// TIA Portal V18 export
DATA_BLOCK "MachineDB"   // DB22
{ S7_Optimized_Access := 'FALSE' }
VERSION : 0.1
// stored: AutoNumber true, DBAccessibleFromOPCUA true, IsOnlyStoredInLoadMemory false, IsWriteProtectedInAS false
   VAR RETAIN
      SerialNumber : Int := 2011;
      AutomateVersion : Int := 6;
      MachineType { ExternalWritable := 'False'} : String := 'ArmadilloV7BR';   // Not writable from HMI
      MachineLimit : Struct
         XSafety : Struct
            PosMax : DInt := 0;
            PosMin : DInt := 0;
            SafetyMargin : DInt;
            VelocityMax : DInt;
            VelocityMin : DInt;
         END_STRUCT;
         YSafety : Struct
            PosMax : DInt := 0;
            PosMin : DInt := 0;
            SafetyMargin : DInt;
            VelocityMax : DInt;
            VelocityMin : DInt;
         END_STRUCT;
         Z1Safety : Struct
            PosMax : DInt := 0;
            PosMin : DInt := 0;
            SafetyMargin : DInt;
            VelocityMax : DInt;
            VelocityMin : DInt;
         END_STRUCT;
         Z2Safety : Struct
            PosMax : DInt := 0;
            PosMin : DInt := 0;
            SafetyMargin : DInt;
            VelocityMax : DInt;
            VelocityMin : DInt;
         END_STRUCT;
         Heater : Struct
            FeedboxStart : DInt;
            FeedboxEnd : DInt;
            PrintboxStart : DInt;
            PrintboxEnd : DInt;
         END_STRUCT;
      END_STRUCT;
      ArmadilloOption : Struct
         MachineTypeNext : String := 'ArmadilloV7BR';
         DoorOption { ExternalWritable := 'False'} : Int := 3;   // SAFETY OPTION, ASK BEFORE CHANGING
         DoorOptionNext : Int := 3;
         DepowderingBox : Int;   // 0 if no box; 1 is we use V1 of the box;
         DepowderingBoxNext : Int;   // 0 if no box; 1 is we use V1 of the box;
         ZAxisDriveOption : String := 'CMMT';   // CMMT;CMMS;
         ZAxisDriveOptionNext : String := 'CMMT';   // CMMT;CMMS;
         UVOption : Int := 1;   // 0 means no UV lamp; 1 version of the UV lamp;
         UVOptionNext : Int := 1;   // 0 means no UV lamp; 1 version of the UV lamp;
         StacklightOption : Int := 1;   // 0 means no Stacklight; 1 version of the Stacklight;
         StacklightOptionNext : Int := 1;   // 0 means no Stacklight; 1 version of the Stacklight;
         CappingStationOption : Int := 1;   // 0 means no Capping Station; 1 version of the Capping Station;
         CappingStationOptionNext : Int := 1;   // 0 means no Capping Station; 1 version of the Capping Station;
      END_STRUCT;
      MachineLimitSecondary : Struct
         NoGoZone01 : Struct   // Temporary not used -> go to DepowderingBoxDimensions
            NoGoZone01_Xstart : DInt;   // Start of the No Go Zone for Depowdering Box
            NoGoZone01_Xend : DInt;   // Start of the No Go Zone for Depowdering Box
            NoGoZone01_Ystart : DInt;   // Start of the No Go Zone for Depowdering Box
            NoGoZone01_Yend : DInt;   // End of the No Go Zone for Depowdering Box
            NoGoZone01_Z1start : DInt;   // Start of the No Go Zone for Depowdering Box
            NoGoZone01_Z1end : DInt;   // End of the No Go Zone for Depowdering Box
            NoGoZone01_Z2start : DInt;   // Start of the No Go Zone for Depowdering Box
            NoGoZone01_Z2end : DInt;   // End of the No Go Zone for Depowdering Box
         END_STRUCT;
      END_STRUCT;
      MachineTypeString : Struct
         _sArmadilloDev { ExternalWritable := 'False'} : String := 'ArmadilloDev';   // Not writable from HMI
         _sArmadilloV2 { ExternalWritable := 'False'} : String := 'ArmadilloV2';   // Not writable from HMI
         _sArmadilloBRV2 { ExternalWritable := 'False'} : String := 'ArmadilloBRV2';   // Not writable from HMI
         _sArmadilloXLV2 { ExternalWritable := 'False'} : String := 'ArmadilloXLV2';   // Not writable from HMI
         _sArmadilloXLBRV2 { ExternalWritable := 'False'} : String := 'ArmadilloXLBRV2';   // Not writable from HMI
         _sArmadilloV6 { ExternalWritable := 'False'} : String := 'ArmadilloV6';   // Machine 2007;
         _sArmadilloV6BR { ExternalWritable := 'False'} : String := 'ArmadilloV6BR';   // Machine 2007;
         _sArmadilloV7 : String := 'ArmadilloV7';   // Machine 2009; 2011;
         _sArmadilloV7BR : String := 'ArmadilloV7BR';   // Machine 2009; 2011;
         _sArmadilloXLV7 : String := 'ArmadilloXLV7';   // Machine 2010;
         _sArmadilloXLV7BR : String := 'ArmadilloXLV7BR';   // Machine 2010;
      END_STRUCT;
      ArmadilloDevMachine : Struct   // Software limit for the Armadillo Dev machine
         XSafety : Struct
            PosMax : DInt := 454000;
            PosMin : DInt := -3000;
            SafetyMargin : DInt := 0;
            VelocityMax : DInt := 500;
            VelocityMin : DInt := 0;
         END_STRUCT;
         YSafety : Struct
            PosMax : DInt := 1100000;
            PosMin : DInt := -3000;
            SafetyMargin : DInt := 0;
            VelocityMax : DInt := 500;
            VelocityMin : DInt;
         END_STRUCT;
         Z1Safety : Struct
            PosMax : DInt := 297850;
            PosMin : DInt := -3000;
            SafetyMargin : DInt := 0;
            VelocityMax : DInt := 20;
            VelocityMin : DInt;
         END_STRUCT;
         Z2Safety : Struct
            PosMax : DInt := 297850;
            PosMin : DInt := -3000;
            SafetyMargin : DInt := 0;
            VelocityMax : DInt := 20;
            VelocityMin : DInt;
         END_STRUCT;
         Heater : Struct
            FeedboxStart : DInt := 100000;
            FeedboxEnd : DInt := 400000;
            PrintboxStart : DInt := 300000;
            PrintboxEnd : DInt := 765000;
         END_STRUCT;
      END_STRUCT;
      ArmadilloBRMachine : Struct   // Software limit for the Armadillo Dev machine
         XSafety : Struct
            PosMax : DInt := 454000;
            PosMin : DInt := -3000;
            SafetyMargin : DInt;
            VelocityMax : DInt;
            VelocityMin : DInt;
         END_STRUCT;
         YSafety : Struct
            PosMax : DInt := 1100000;
            PosMin : DInt := -3000;
            SafetyMargin : DInt;
            VelocityMax : DInt;
            VelocityMin : DInt;
         END_STRUCT;
         Z1Safety : Struct
            PosMax : DInt := 94000;   // v1 = 210500
            PosMin : DInt := -3000;
            SafetyMargin : DInt;
            VelocityMax : DInt;
            VelocityMin : DInt;
         END_STRUCT;
         Z2Safety : Struct
            PosMax : DInt := 94000;   // v1 = 210500
            PosMin : DInt := -3000;
            SafetyMargin : DInt;
            VelocityMax : DInt;
            VelocityMin : DInt;
         END_STRUCT;
         Heater : Struct
            FeedboxStart : DInt;
            FeedboxEnd : DInt;
            PrintboxStart : DInt;
            PrintboxEnd : DInt;
         END_STRUCT;
      END_STRUCT;
      ArmadilloXLMachine : Struct   // Software limit for the Armadillo Production machine
         XSafety : Struct
            PosMax : DInt := 516000;
            PosMin : DInt := -3000;
            SafetyMargin : DInt;
            VelocityMax : DInt;
            VelocityMin : DInt;
         END_STRUCT;
         YSafety : Struct
            PosMax : DInt := 1380000;
            PosMin : DInt := -3000;
            SafetyMargin : DInt;
            VelocityMax : DInt;
            VelocityMin : DInt;
         END_STRUCT;
         Z1Safety : Struct
            PosMax : DInt := 302000;
            PosMin : DInt := -500;
            SafetyMargin : DInt;
            VelocityMax : DInt;
            VelocityMin : DInt;
         END_STRUCT;
         Z2Safety : Struct
            PosMax : DInt := 302000;
            PosMin : DInt := -500;
            SafetyMargin : DInt;
            VelocityMax : DInt;
            VelocityMin : DInt;
         END_STRUCT;
         Heater : Struct
            FeedboxStart : DInt;
            FeedboxEnd : DInt;
            PrintboxStart : DInt;
            PrintboxEnd : DInt;
         END_STRUCT;
      END_STRUCT;
      ArmadilloXLBRMachine : Struct   // Software limit for the Armadillo Production machine
         XSafety : Struct
            PosMax : DInt := 516000;
            PosMin : DInt := -3000;
            SafetyMargin : DInt;
            VelocityMax : DInt;
            VelocityMin : DInt;
         END_STRUCT;
         YSafety : Struct
            PosMax : DInt := 1380000;
            PosMin : DInt := -3000;
            SafetyMargin : DInt;
            VelocityMax : DInt;
            VelocityMin : DInt;
         END_STRUCT;
         Z1Safety : Struct
            PosMax : DInt := 210500;
            PosMin : DInt := -3000;
            SafetyMargin : DInt;
            VelocityMax : DInt;
            VelocityMin : DInt;
         END_STRUCT;
         Z2Safety : Struct
            PosMax : DInt := 210500;
            PosMin : DInt := -3000;
            SafetyMargin : DInt;
            VelocityMax : DInt;
            VelocityMin : DInt;
         END_STRUCT;
         Heater : Struct
            FeedboxStart : DInt;
            FeedboxEnd : DInt;
            PrintboxStart : DInt;
            PrintboxEnd : DInt;
         END_STRUCT;
      END_STRUCT;
      ArmadilloV6Machine : Struct   // 2007 Eurostar Software limit for the Armadillo V6 machine
         XSafety : Struct
            PosMax : DInt := 500000;
            PosMin : DInt := 0;
            SafetyMargin : DInt := 5000;
            VelocityMax : DInt := 500;
            VelocityMin : DInt := 0;
         END_STRUCT;
         YSafety : Struct
            PosMax : DInt := 1365000;
            PosMin : DInt := 0;
            SafetyMargin : DInt := 5000;
            VelocityMax : DInt := 500;
            VelocityMin : DInt;
         END_STRUCT;
         Z1Safety : Struct
            PosMax : DInt := 300000;
            PosMin : DInt := 0;
            SafetyMargin : DInt := 2000;
            VelocityMax : DInt;
            VelocityMin : DInt;
         END_STRUCT;
         Z2Safety : Struct
            PosMax : DInt := 300000;
            PosMin : DInt := 0;
            SafetyMargin : DInt := 2000;
            VelocityMax : DInt;
            VelocityMin : DInt;
         END_STRUCT;
         Heater : Struct
            FeedboxStart : DInt := 270000;
            FeedboxEnd : DInt := 580000;
            PrintboxStart : DInt := 580000;
            PrintboxEnd : DInt := 880000;
         END_STRUCT;
      END_STRUCT;
      ArmadilloV6BRMachine : Struct   // 2007 Eurostar Software limit for the Armadillo V6 Bed Reduction machine
         XSafety : Struct
            PosMax : DInt := 500000;
            PosMin : DInt := 0;
            SafetyMargin : DInt := 5000;
            VelocityMax : DInt := 500;
            VelocityMin : DInt;
         END_STRUCT;
         YSafety : Struct
            PosMax : DInt := 1365000;
            PosMin : DInt := 0;
            SafetyMargin : DInt := 5000;
            VelocityMax : DInt := 500;
            VelocityMin : DInt;
         END_STRUCT;
         Z1Safety : Struct
            PosMax : DInt := 90000;   // v1 = 210500
            PosMin : DInt := 0;
            SafetyMargin : DInt := 2000;
            VelocityMax : DInt;
            VelocityMin : DInt;
         END_STRUCT;
         Z2Safety : Struct
            PosMax : DInt := 90000;   // v1 = 210500
            PosMin : DInt := 0;
            SafetyMargin : DInt := 2000;
            VelocityMax : DInt;
            VelocityMin : DInt;
         END_STRUCT;
         Heater : Struct
            FeedboxStart : DInt := 470000;
            FeedboxEnd : DInt := 580000;
            PrintboxStart : DInt := 580000;
            PrintboxEnd : DInt := 680000;
         END_STRUCT;
      END_STRUCT;
      ArmadilloV7Machine : Struct   // 2009, 2011 Normal Software limit for the Armadillo V6 machine
         XSafety : Struct
            PosMax : DInt := 435000;
            PosMin : DInt := -3000;
            SafetyMargin : DInt := 5000;
            VelocityMax : DInt := 500;
            VelocityMin : DInt := 0;
         END_STRUCT;
         YSafety : Struct
            PosMax : DInt := 1065000;
            PosMin : DInt := -3000;
            SafetyMargin : DInt := 5000;
            VelocityMax : DInt := 500;
            VelocityMin : DInt;
         END_STRUCT;
         Z1Safety : Struct
            PosMax : DInt := 312000;
            PosMin : DInt := 0;
            SafetyMargin : DInt := 2000;
            VelocityMax : DInt;
            VelocityMin : DInt;
         END_STRUCT;
         Z2Safety : Struct
            PosMax : DInt := 312000;
            PosMin : DInt := 0;
            SafetyMargin : DInt := 2000;
            VelocityMax : DInt;
            VelocityMin : DInt;
         END_STRUCT;
         Heater : Struct
            FeedboxStart : DInt := 100000;
            FeedboxEnd : DInt := 430000;
            PrintboxStart : DInt := 430000;
            PrintboxEnd : DInt := 740000;
         END_STRUCT;
      END_STRUCT;
      ArmadilloV7BRMachine : Struct   // 2009, 2011 Normal Software limit for the Armadillo V6 Bed Reduction machine
         XSafety : Struct
            PosMax : DInt := 435000;
            PosMin : DInt := -3000;
            SafetyMargin : DInt := 5000;
            VelocityMax : DInt := 500;
            VelocityMin : DInt;
         END_STRUCT;
         YSafety : Struct
            PosMax : DInt := 1065000;
            PosMin : DInt := -3000;
            SafetyMargin : DInt := 5000;
            VelocityMax : DInt := 500;
            VelocityMin : DInt;
         END_STRUCT;
         Z1Safety : Struct
            PosMax : DInt := 86000;
            PosMin : DInt := 0;
            SafetyMargin : DInt := 2000;
            VelocityMax : DInt;
            VelocityMin : DInt;
         END_STRUCT;
         Z2Safety : Struct
            PosMax : DInt := 86000;
            PosMin : DInt := 0;
            SafetyMargin : DInt := 2000;
            VelocityMax : DInt;
            VelocityMin : DInt;
         END_STRUCT;
         Heater : Struct
            FeedboxStart : DInt := 250000;
            FeedboxEnd : DInt := 360000;
            PrintboxStart : DInt := 360000;
            PrintboxEnd : DInt := 490000;
         END_STRUCT;
      END_STRUCT;
      ArmadilloXLV7Machine : Struct   // 2010 XL Software limit for the Armadillo V6 machine
         XSafety : Struct
            PosMax : DInt := 500000;
            PosMin : DInt := -3000;
            SafetyMargin : DInt := 5000;
            VelocityMax : DInt := 500;
            VelocityMin : DInt := 0;
         END_STRUCT;
         YSafety : Struct
            PosMax : DInt := 1365000;
            PosMin : DInt := -3000;
            SafetyMargin : DInt := 5000;
            VelocityMax : DInt := 500;
            VelocityMin : DInt;
         END_STRUCT;
         Z1Safety : Struct
            PosMax : DInt := 312000;
            PosMin : DInt := 0;
            SafetyMargin : DInt := 2000;
            VelocityMax : DInt;
            VelocityMin : DInt;
         END_STRUCT;
         Z2Safety : Struct
            PosMax : DInt := 312000;
            PosMin : DInt := 0;
            SafetyMargin : DInt := 2000;
            VelocityMax : DInt;
            VelocityMin : DInt;
         END_STRUCT;
         Heater : Struct
            FeedboxStart : DInt := 150000;
            FeedboxEnd : DInt := 610000;
            PrintboxStart : DInt := 610000;
            PrintboxEnd : DInt := 1100000;
         END_STRUCT;
      END_STRUCT;
      ArmadilloXLV7BRMachine : Struct   // 2010 XL Software limit for the Armadillo V6 Bed Reduction machine
         XSafety : Struct
            PosMax : DInt := 500000;
            PosMin : DInt := -3000;
            SafetyMargin : DInt := 5000;
            VelocityMax : DInt := 500;
            VelocityMin : DInt;
         END_STRUCT;
         YSafety : Struct
            PosMax : DInt := 1365000;
            PosMin : DInt := -3000;
            SafetyMargin : DInt := 5000;
            VelocityMax : DInt := 500;
            VelocityMin : DInt;
         END_STRUCT;
         Z1Safety : Struct
            PosMax : DInt := 86000;
            PosMin : DInt := 0;
            SafetyMargin : DInt := 2000;
            VelocityMax : DInt;
            VelocityMin : DInt;
         END_STRUCT;
         Z2Safety : Struct
            PosMax : DInt := 86000;
            PosMin : DInt := 0;
            SafetyMargin : DInt := 2000;
            VelocityMax : DInt;
            VelocityMin : DInt;
         END_STRUCT;
         Heater : Struct
            FeedboxStart : DInt := 440000;
            FeedboxEnd : DInt := 620000;
            PrintboxStart : DInt := 620000;
            PrintboxEnd : DInt := 770000;
         END_STRUCT;
      END_STRUCT;
      DepowderingBoxDimensions : Struct   // Should be integrated with machine limits in the future
         DepowderingBoxHeight : DInt := 27000;
         DepowderingBoxWidth : DInt := 0;
         DepowderingBoxMargin : DInt := 3000;
         DepowderingBoxNormal : Struct
            DepowderingBoxNormalXstart : DInt := 0;
            DepowderingBoxNormalXend : DInt := 550000;
            DepowderingBoxNormalYstart : DInt := 180000;
            DepowderingBoxNormalYend : DInt := 1500000;
         END_STRUCT;
         DepowderingBoxXL : Struct
            DepowderingBoxXLXstart : DInt := 0;
            DepowderingBoxXLXend : DInt := 550000;
            DepowderingBoxXLYstart : DInt := 190000;
            DepowderingBoxXLYend : DInt := 1500000;
         END_STRUCT;
      END_STRUCT;
   END_VAR
BEGIN
END_DATA_BLOCK
